// TIA Portal V17 export
// export: Created 2024-08-07T21:43:58.5559436Z, ExportSetting WithDefaults, DisplayName Totally Integrated Automation Portal, DisplayVersion V17 Update 7, DisplayName TIA Portal Openness, DisplayVersion V17 Update 7, DisplayName TIA Portal Version Control Interface, DisplayVersion V17, DisplayName SINAMICS Startdrive Advanced, DisplayVersion V17 SP2, DisplayName SINAMICS Startdrive G110M, G120, G120C, G120D, G120P, G115D, DisplayVersion V17 SP2, DisplayName SINAMICS Startdrive G130, G150, S120, S150, SINAMICS MV, S210, DisplayVersion V17 SP2, DisplayName STEP 7 Professional, DisplayVersion V17 Update 7, DisplayName STEP 7 Safety, DisplayVersion V17 Update 6, DisplayName WinCC Advanced / Unified PC, DisplayVersion V17 Update 7
FUNCTION "READERS" : Void   // FC19, LAD
{ S7_Optimized_Access := 'TRUE' }
VERSION : 0.1
// stored: AutoNumber true, IsIECCheckEnabled false, SetENOAutomatically false, UDAEnableTagReadback false
   VAR_TEMP
      done1 : Bool;
      done2 : Bool;
      done3 : Bool;
      done4 : Bool;
      ERROR_RECIBIDO_ESCANER_REAR_TUBE : Int;
      ERROR_RECIBIDO_ESCANER_FRONT_TUBE : Int;
      ERROR_RECIBIDO_ESCANER_LH_MEMBER : Int;
      ERROR_RECIBIDO_ESCANER_RH_MEMBER : Int;
   END_VAR
   VAR_TEMP   // added for the SCL form of the ladder/FBD networks
      _w1 : Bool;
   END_VAR
BEGIN

REGION Network 1: INIT
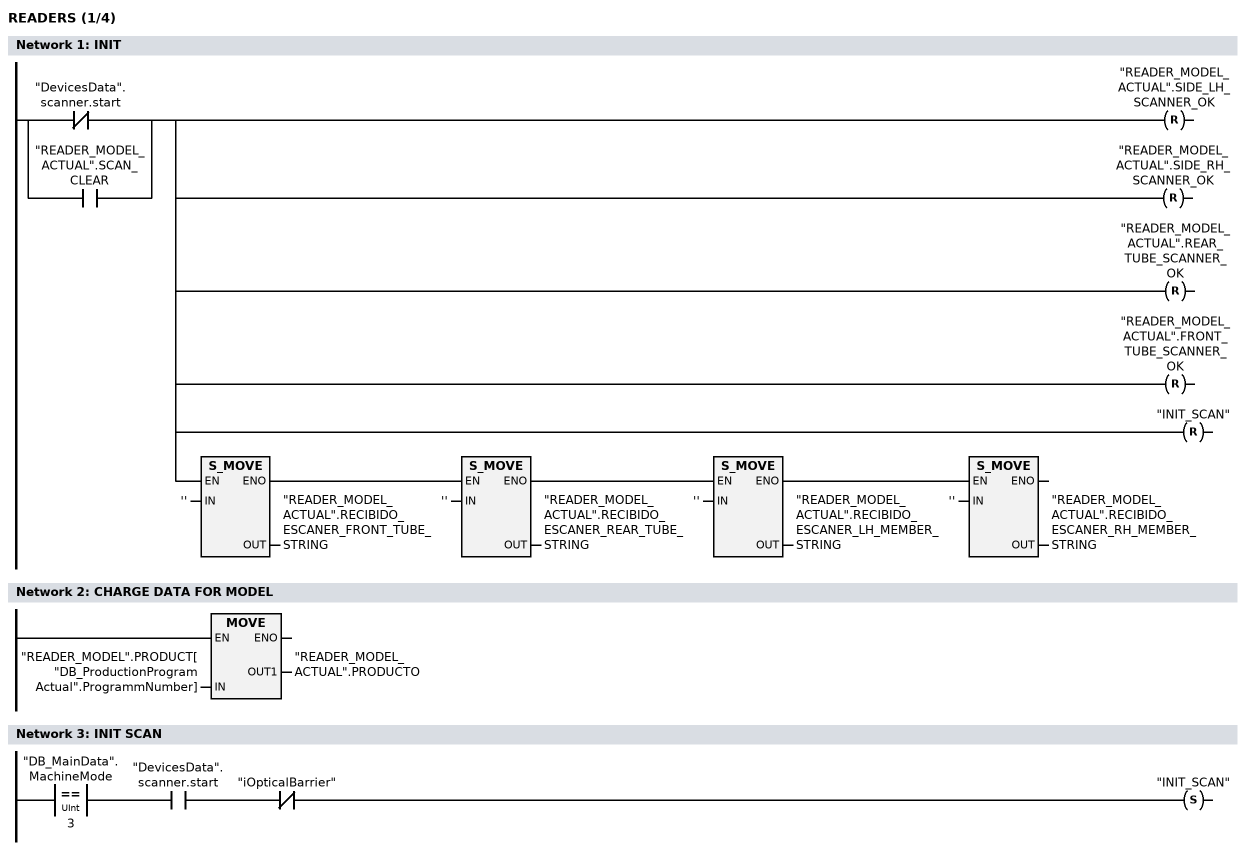
   RUNG wire#powerrail
      I_Contact( "DevicesData".scanner.start )
      wire#w1
      R_Coil( "READER_MODEL_ACTUAL".SIDE_LH_SCANNER_OK )
   END_RUNG
   RUNG wire#powerrail
      Contact( "READER_MODEL_ACTUAL".SCAN_CLEAR )
   END_RUNG wire#w1
   RUNG wire#w1
      R_Coil( "READER_MODEL_ACTUAL".SIDE_RH_SCANNER_OK )
   END_RUNG
   RUNG wire#w1
      R_Coil( "READER_MODEL_ACTUAL".REAR_TUBE_SCANNER_OK )
   END_RUNG
   RUNG wire#w1
      R_Coil( "READER_MODEL_ACTUAL".FRONT_TUBE_SCANNER_OK )
   END_RUNG
   RUNG wire#w1
      R_Coil( "INIT_SCAN" )
   END_RUNG
   RUNG wire#w1
      S_Move(in := '', out => "READER_MODEL_ACTUAL".RECIBIDO_ESCANER_FRONT_TUBE_STRING)
      S_Move(in := '', out => "READER_MODEL_ACTUAL".RECIBIDO_ESCANER_REAR_TUBE_STRING)
      S_Move(in := '', out => "READER_MODEL_ACTUAL".RECIBIDO_ESCANER_LH_MEMBER_STRING)
      S_Move(in := '', out => "READER_MODEL_ACTUAL".RECIBIDO_ESCANER_RH_MEMBER_STRING)
   END_RUNG
   // the same network as SCL:
   IF NOT "DevicesData".scanner.start OR "READER_MODEL_ACTUAL".SCAN_CLEAR THEN
       "READER_MODEL_ACTUAL".SIDE_LH_SCANNER_OK := FALSE;
       "READER_MODEL_ACTUAL".SIDE_RH_SCANNER_OK := FALSE;
       "READER_MODEL_ACTUAL".REAR_TUBE_SCANNER_OK := FALSE;
       "READER_MODEL_ACTUAL".FRONT_TUBE_SCANNER_OK := FALSE;
       "INIT_SCAN" := FALSE;
       "READER_MODEL_ACTUAL".RECIBIDO_ESCANER_FRONT_TUBE_STRING := '';
       "READER_MODEL_ACTUAL".RECIBIDO_ESCANER_REAR_TUBE_STRING := '';
       "READER_MODEL_ACTUAL".RECIBIDO_ESCANER_LH_MEMBER_STRING := '';
       "READER_MODEL_ACTUAL".RECIBIDO_ESCANER_RH_MEMBER_STRING := '';
   END_IF;
END_REGION

REGION Network 2: CHARGE DATA FOR MODEL
   RUNG wire#powerrail
      Move(in := "READER_MODEL".PRODUCT["DB_ProductionProgramActual".ProgrammNumber], out1 => "READER_MODEL_ACTUAL".PRODUCTO)
   END_RUNG
   // the same network as SCL:
   "READER_MODEL_ACTUAL".PRODUCTO := "READER_MODEL".PRODUCT["DB_ProductionProgramActual".ProgrammNumber];
END_REGION

REGION Network 3: INIT SCAN
   RUNG wire#powerrail
      { S7_Templates := "SrcType := UInt" } EQ_Contact(in1 := "DB_MainData".MachineMode, in2 := 3)
      Contact( "DevicesData".scanner.start )
      I_Contact( "iOpticalBarrier" )
      S_Coil( "INIT_SCAN" )
   END_RUNG
   // the same network as SCL:
   IF ("DB_MainData".MachineMode = 3) AND "DevicesData".scanner.start AND NOT "iOpticalBarrier" THEN
       "INIT_SCAN" := TRUE;
   END_IF;
END_REGION

REGION Network 4: LECTURA ESCANER REAR TUBE
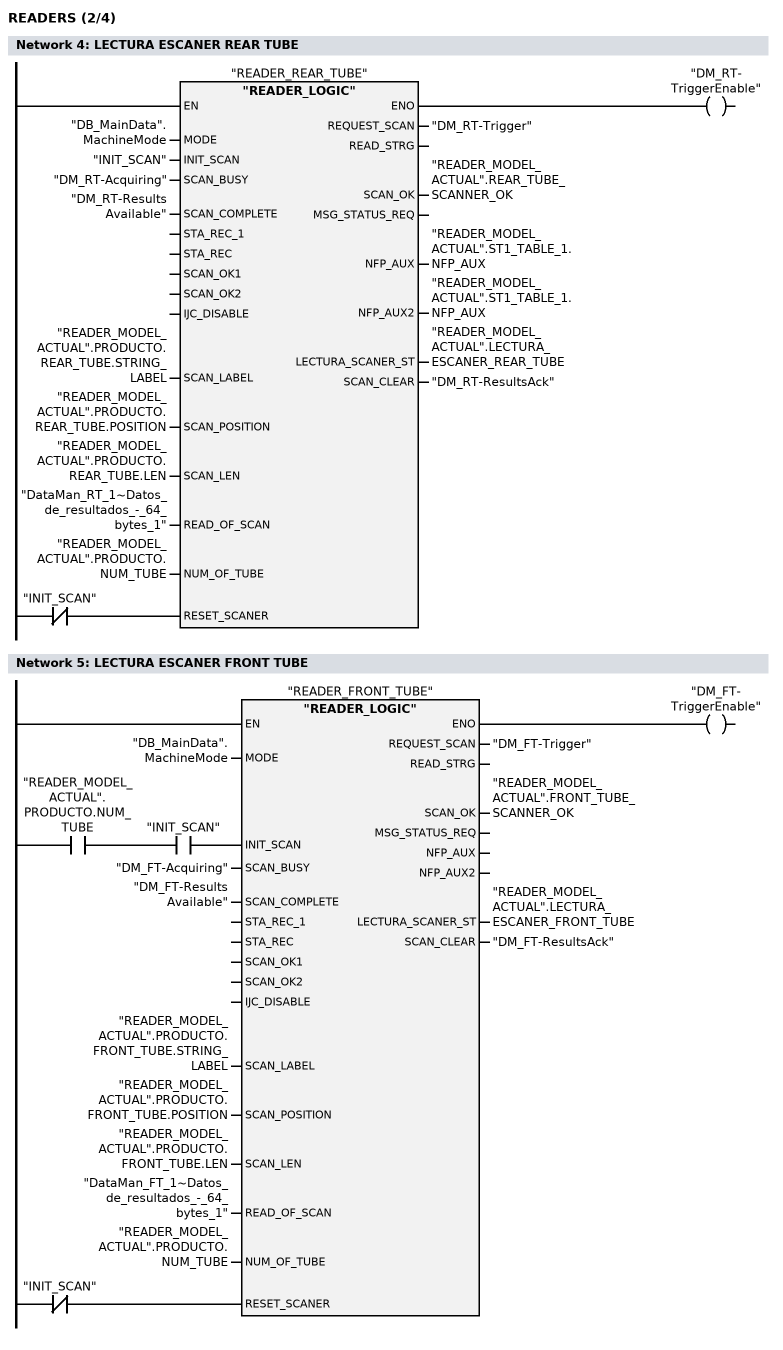
   RUNG wire#powerrail
      "READER_REAR_TUBE"(RESET_SCANER := wire#w1, MODE := "DB_MainData".MachineMode, INIT_SCAN := "INIT_SCAN", SCAN_BUSY := "DM_RT-Acquiring", SCAN_COMPLETE := "DM_RT-Results Available", STA_REC_1 :=, STA_REC :=, SCAN_OK1 :=, SCAN_OK2 :=, IJC_DISABLE :=, SCAN_LABEL := "READER_MODEL_ACTUAL".PRODUCTO.REAR_TUBE.STRING_LABEL, SCAN_POSITION := "READER_MODEL_ACTUAL".PRODUCTO.REAR_TUBE.POSITION, SCAN_LEN := "READER_MODEL_ACTUAL".PRODUCTO.REAR_TUBE.LEN, READ_OF_SCAN := "DataMan_RT_1~Datos_de_resultados_-_64_bytes_1", NUM_OF_TUBE := "READER_MODEL_ACTUAL".PRODUCTO.NUM_TUBE, REQUEST_SCAN => "DM_RT-Trigger", READ_STRG =>, SCAN_OK => "READER_MODEL_ACTUAL".REAR_TUBE_SCANNER_OK, MSG_STATUS_REQ =>, NFP_AUX => "READER_MODEL_ACTUAL".ST1_TABLE_1.NFP_AUX, NFP_AUX2 => "READER_MODEL_ACTUAL".ST1_TABLE_1.NFP_AUX, LECTURA_SCANER_ST => "READER_MODEL_ACTUAL".LECTURA_ESCANER_REAR_TUBE, SCAN_CLEAR => "DM_RT-ResultsAck")
      Coil( "DM_RT-TriggerEnable" )
   END_RUNG
   RUNG wire#powerrail
      I_Contact( "INIT_SCAN" )
   END_RUNG wire#w1
   // the same network as SCL:
   "READER_REAR_TUBE"(MODE := "DB_MainData".MachineMode,   // "READER_LOGIC"
                      INIT_SCAN := "INIT_SCAN",
                      SCAN_BUSY := "DM_RT-Acquiring",
                      SCAN_COMPLETE := "DM_RT-Results Available",
                      SCAN_LABEL := "READER_MODEL_ACTUAL".PRODUCTO.REAR_TUBE.STRING_LABEL,
                      SCAN_POSITION := "READER_MODEL_ACTUAL".PRODUCTO.REAR_TUBE.POSITION,
                      SCAN_LEN := "READER_MODEL_ACTUAL".PRODUCTO.REAR_TUBE.LEN,
                      READ_OF_SCAN := "DataMan_RT_1~Datos_de_resultados_-_64_bytes_1",
                      NUM_OF_TUBE := "READER_MODEL_ACTUAL".PRODUCTO.NUM_TUBE,
                      RESET_SCANER := NOT "INIT_SCAN",
                      REQUEST_SCAN => "DM_RT-Trigger",
                      SCAN_OK => "READER_MODEL_ACTUAL".REAR_TUBE_SCANNER_OK,
                      NFP_AUX => "READER_MODEL_ACTUAL".ST1_TABLE_1.NFP_AUX,
                      NFP_AUX2 => "READER_MODEL_ACTUAL".ST1_TABLE_1.NFP_AUX,
                      LECTURA_SCANER_ST => "READER_MODEL_ACTUAL".LECTURA_ESCANER_REAR_TUBE,
                      SCAN_CLEAR => "DM_RT-ResultsAck",
                      ENO => #_w1);
   "DM_RT-TriggerEnable" := #_w1;
END_REGION

REGION Network 5: LECTURA ESCANER FRONT TUBE
   RUNG wire#powerrail
      "READER_FRONT_TUBE"(INIT_SCAN := wire#w1, RESET_SCANER := wire#w2, MODE := "DB_MainData".MachineMode, SCAN_BUSY := "DM_FT-Acquiring", SCAN_COMPLETE := "DM_FT-Results Available", STA_REC_1 :=, STA_REC :=, SCAN_OK1 :=, SCAN_OK2 :=, IJC_DISABLE :=, SCAN_LABEL := "READER_MODEL_ACTUAL".PRODUCTO.FRONT_TUBE.STRING_LABEL, SCAN_POSITION := "READER_MODEL_ACTUAL".PRODUCTO.FRONT_TUBE.POSITION, SCAN_LEN := "READER_MODEL_ACTUAL".PRODUCTO.FRONT_TUBE.LEN, READ_OF_SCAN := "DataMan_FT_1~Datos_de_resultados_-_64_bytes_1", NUM_OF_TUBE := "READER_MODEL_ACTUAL".PRODUCTO.NUM_TUBE, REQUEST_SCAN => "DM_FT-Trigger", READ_STRG =>, SCAN_OK => "READER_MODEL_ACTUAL".FRONT_TUBE_SCANNER_OK, MSG_STATUS_REQ =>, NFP_AUX =>, NFP_AUX2 =>, LECTURA_SCANER_ST => "READER_MODEL_ACTUAL".LECTURA_ESCANER_FRONT_TUBE, SCAN_CLEAR => "DM_FT-ResultsAck")
      Coil( "DM_FT-TriggerEnable" )
   END_RUNG
   RUNG wire#powerrail
      Contact( "READER_MODEL_ACTUAL".PRODUCTO.NUM_TUBE )
      Contact( "INIT_SCAN" )
   END_RUNG wire#w1
   RUNG wire#powerrail
      I_Contact( "INIT_SCAN" )
   END_RUNG wire#w2
   // the same network as SCL:
   "READER_FRONT_TUBE"(MODE := "DB_MainData".MachineMode,   // "READER_LOGIC"
                       INIT_SCAN := "READER_MODEL_ACTUAL".PRODUCTO.NUM_TUBE AND "INIT_SCAN",
                       SCAN_BUSY := "DM_FT-Acquiring",
                       SCAN_COMPLETE := "DM_FT-Results Available",
                       SCAN_LABEL := "READER_MODEL_ACTUAL".PRODUCTO.FRONT_TUBE.STRING_LABEL,
                       SCAN_POSITION := "READER_MODEL_ACTUAL".PRODUCTO.FRONT_TUBE.POSITION,
                       SCAN_LEN := "READER_MODEL_ACTUAL".PRODUCTO.FRONT_TUBE.LEN,
                       READ_OF_SCAN := "DataMan_FT_1~Datos_de_resultados_-_64_bytes_1",
                       NUM_OF_TUBE := "READER_MODEL_ACTUAL".PRODUCTO.NUM_TUBE,
                       RESET_SCANER := NOT "INIT_SCAN",
                       REQUEST_SCAN => "DM_FT-Trigger",
                       SCAN_OK => "READER_MODEL_ACTUAL".FRONT_TUBE_SCANNER_OK,
                       LECTURA_SCANER_ST => "READER_MODEL_ACTUAL".LECTURA_ESCANER_FRONT_TUBE,
                       SCAN_CLEAR => "DM_FT-ResultsAck",
                       ENO => #_w1);
   "DM_FT-TriggerEnable" := #_w1;
END_REGION

REGION Network 6: LECTURA ESCANER SIDE LH
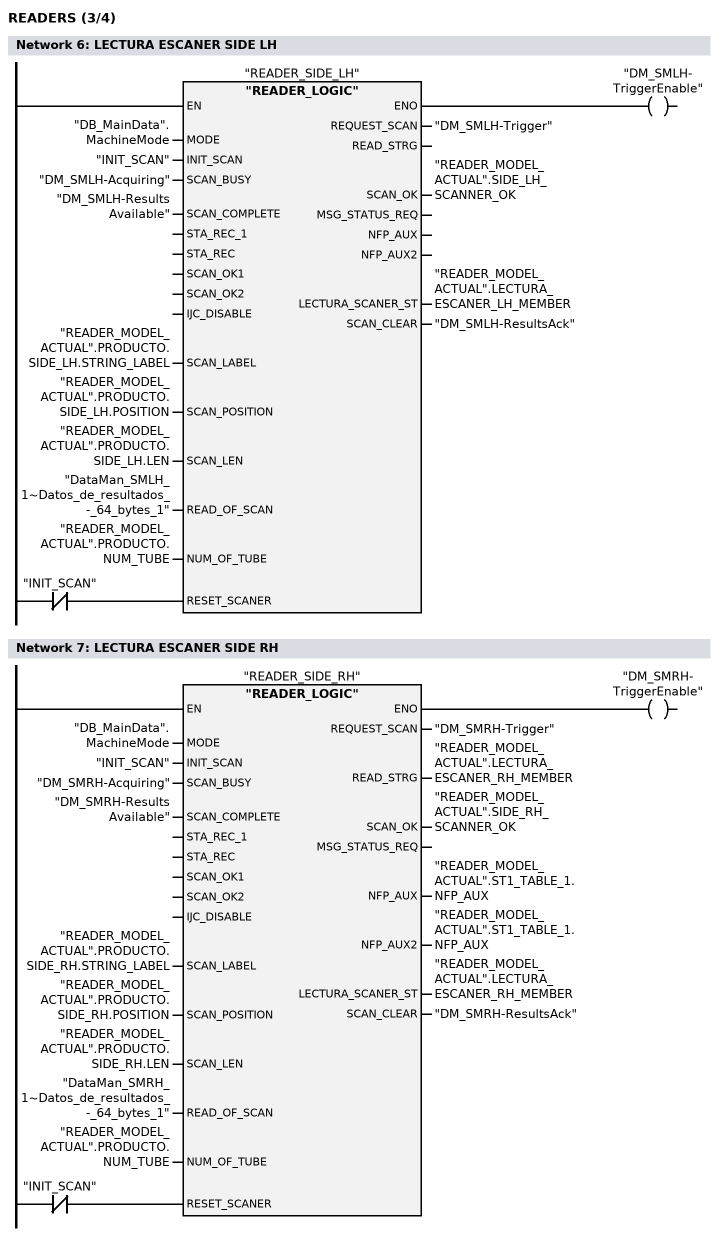
   RUNG wire#powerrail
      "READER_SIDE_LH"(RESET_SCANER := wire#w1, MODE := "DB_MainData".MachineMode, INIT_SCAN := "INIT_SCAN", SCAN_BUSY := "DM_SMLH-Acquiring", SCAN_COMPLETE := "DM_SMLH-Results Available", STA_REC_1 :=, STA_REC :=, SCAN_OK1 :=, SCAN_OK2 :=, IJC_DISABLE :=, SCAN_LABEL := "READER_MODEL_ACTUAL".PRODUCTO.SIDE_LH.STRING_LABEL, SCAN_POSITION := "READER_MODEL_ACTUAL".PRODUCTO.SIDE_LH.POSITION, SCAN_LEN := "READER_MODEL_ACTUAL".PRODUCTO.SIDE_LH.LEN, READ_OF_SCAN := "DataMan_SMLH_1~Datos_de_resultados_-_64_bytes_1", NUM_OF_TUBE := "READER_MODEL_ACTUAL".PRODUCTO.NUM_TUBE, REQUEST_SCAN => "DM_SMLH-Trigger", READ_STRG =>, SCAN_OK => "READER_MODEL_ACTUAL".SIDE_LH_SCANNER_OK, MSG_STATUS_REQ =>, NFP_AUX =>, NFP_AUX2 =>, LECTURA_SCANER_ST => "READER_MODEL_ACTUAL".LECTURA_ESCANER_LH_MEMBER, SCAN_CLEAR => "DM_SMLH-ResultsAck")
      Coil( "DM_SMLH-TriggerEnable" )
   END_RUNG
   RUNG wire#powerrail
      I_Contact( "INIT_SCAN" )
   END_RUNG wire#w1
   // the same network as SCL:
   "READER_SIDE_LH"(MODE := "DB_MainData".MachineMode,   // "READER_LOGIC"
                    INIT_SCAN := "INIT_SCAN",
                    SCAN_BUSY := "DM_SMLH-Acquiring",
                    SCAN_COMPLETE := "DM_SMLH-Results Available",
                    SCAN_LABEL := "READER_MODEL_ACTUAL".PRODUCTO.SIDE_LH.STRING_LABEL,
                    SCAN_POSITION := "READER_MODEL_ACTUAL".PRODUCTO.SIDE_LH.POSITION,
                    SCAN_LEN := "READER_MODEL_ACTUAL".PRODUCTO.SIDE_LH.LEN,
                    READ_OF_SCAN := "DataMan_SMLH_1~Datos_de_resultados_-_64_bytes_1",
                    NUM_OF_TUBE := "READER_MODEL_ACTUAL".PRODUCTO.NUM_TUBE,
                    RESET_SCANER := NOT "INIT_SCAN",
                    REQUEST_SCAN => "DM_SMLH-Trigger",
                    SCAN_OK => "READER_MODEL_ACTUAL".SIDE_LH_SCANNER_OK,
                    LECTURA_SCANER_ST => "READER_MODEL_ACTUAL".LECTURA_ESCANER_LH_MEMBER,
                    SCAN_CLEAR => "DM_SMLH-ResultsAck",
                    ENO => #_w1);
   "DM_SMLH-TriggerEnable" := #_w1;
END_REGION

REGION Network 7: LECTURA ESCANER SIDE RH
   RUNG wire#powerrail
      "READER_SIDE_RH"(RESET_SCANER := wire#w1, MODE := "DB_MainData".MachineMode, INIT_SCAN := "INIT_SCAN", SCAN_BUSY := "DM_SMRH-Acquiring", SCAN_COMPLETE := "DM_SMRH-Results Available", STA_REC_1 :=, STA_REC :=, SCAN_OK1 :=, SCAN_OK2 :=, IJC_DISABLE :=, SCAN_LABEL := "READER_MODEL_ACTUAL".PRODUCTO.SIDE_RH.STRING_LABEL, SCAN_POSITION := "READER_MODEL_ACTUAL".PRODUCTO.SIDE_RH.POSITION, SCAN_LEN := "READER_MODEL_ACTUAL".PRODUCTO.SIDE_RH.LEN, READ_OF_SCAN := "DataMan_SMRH_1~Datos_de_resultados_-_64_bytes_1", NUM_OF_TUBE := "READER_MODEL_ACTUAL".PRODUCTO.NUM_TUBE, REQUEST_SCAN => "DM_SMRH-Trigger", READ_STRG => "READER_MODEL_ACTUAL".LECTURA_ESCANER_RH_MEMBER, SCAN_OK => "READER_MODEL_ACTUAL".SIDE_RH_SCANNER_OK, MSG_STATUS_REQ =>, NFP_AUX => "READER_MODEL_ACTUAL".ST1_TABLE_1.NFP_AUX, NFP_AUX2 => "READER_MODEL_ACTUAL".ST1_TABLE_1.NFP_AUX, LECTURA_SCANER_ST => "READER_MODEL_ACTUAL".LECTURA_ESCANER_RH_MEMBER, SCAN_CLEAR => "DM_SMRH-ResultsAck")
      Coil( "DM_SMRH-TriggerEnable" )
   END_RUNG
   RUNG wire#powerrail
      I_Contact( "INIT_SCAN" )
   END_RUNG wire#w1
   // the same network as SCL:
   "READER_SIDE_RH"(MODE := "DB_MainData".MachineMode,   // "READER_LOGIC"
                    INIT_SCAN := "INIT_SCAN",
                    SCAN_BUSY := "DM_SMRH-Acquiring",
                    SCAN_COMPLETE := "DM_SMRH-Results Available",
                    SCAN_LABEL := "READER_MODEL_ACTUAL".PRODUCTO.SIDE_RH.STRING_LABEL,
                    SCAN_POSITION := "READER_MODEL_ACTUAL".PRODUCTO.SIDE_RH.POSITION,
                    SCAN_LEN := "READER_MODEL_ACTUAL".PRODUCTO.SIDE_RH.LEN,
                    READ_OF_SCAN := "DataMan_SMRH_1~Datos_de_resultados_-_64_bytes_1",
                    NUM_OF_TUBE := "READER_MODEL_ACTUAL".PRODUCTO.NUM_TUBE,
                    RESET_SCANER := NOT "INIT_SCAN",
                    REQUEST_SCAN => "DM_SMRH-Trigger",
                    READ_STRG => "READER_MODEL_ACTUAL".LECTURA_ESCANER_RH_MEMBER,
                    SCAN_OK => "READER_MODEL_ACTUAL".SIDE_RH_SCANNER_OK,
                    NFP_AUX => "READER_MODEL_ACTUAL".ST1_TABLE_1.NFP_AUX,
                    NFP_AUX2 => "READER_MODEL_ACTUAL".ST1_TABLE_1.NFP_AUX,
                    LECTURA_SCANER_ST => "READER_MODEL_ACTUAL".LECTURA_ESCANER_RH_MEMBER,
                    SCAN_CLEAR => "DM_SMRH-ResultsAck",
                    ENO => #_w1);
   "DM_SMRH-TriggerEnable" := #_w1;
END_REGION

REGION Network 8: ALL SCANER OK
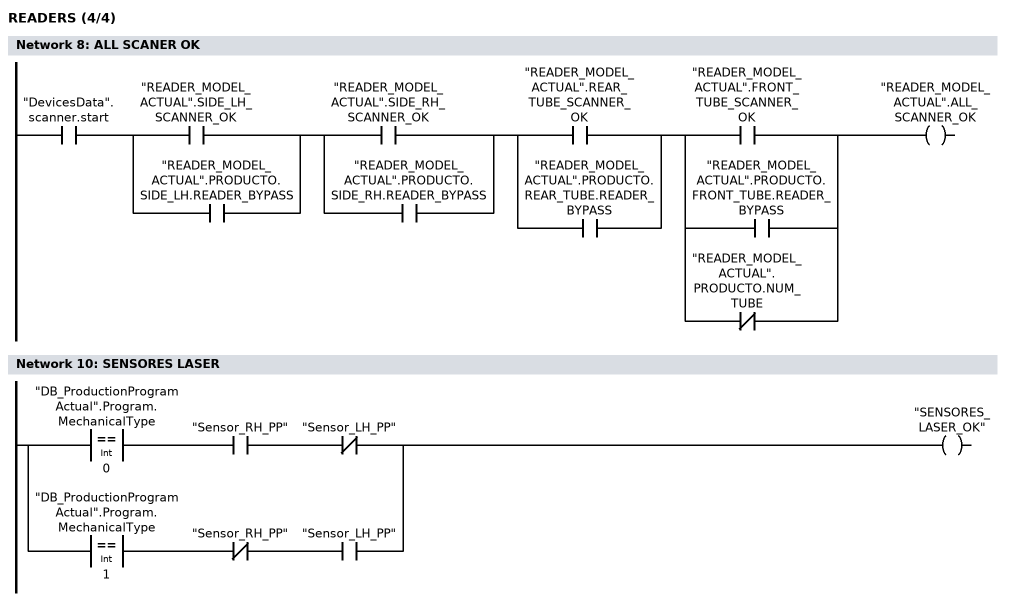
   RUNG wire#powerrail
      Contact( "DevicesData".scanner.start )
      wire#w1
      Contact( "READER_MODEL_ACTUAL".SIDE_LH_SCANNER_OK )
      wire#w2
      Contact( "READER_MODEL_ACTUAL".SIDE_RH_SCANNER_OK )
      wire#w3
      Contact( "READER_MODEL_ACTUAL".REAR_TUBE_SCANNER_OK )
      wire#w4
      Contact( "READER_MODEL_ACTUAL".FRONT_TUBE_SCANNER_OK )
      wire#w5
      Coil( "READER_MODEL_ACTUAL".ALL_SCANNER_OK )
   END_RUNG
   RUNG wire#w1
      Contact( "READER_MODEL_ACTUAL".PRODUCTO.SIDE_LH.READER_BYPASS )
   END_RUNG wire#w2
   RUNG wire#w2
      Contact( "READER_MODEL_ACTUAL".PRODUCTO.SIDE_RH.READER_BYPASS )
   END_RUNG wire#w3
   RUNG wire#w3
      Contact( "READER_MODEL_ACTUAL".PRODUCTO.REAR_TUBE.READER_BYPASS )
   END_RUNG wire#w4
   RUNG wire#w4
      Contact( "READER_MODEL_ACTUAL".PRODUCTO.FRONT_TUBE.READER_BYPASS )
   END_RUNG wire#w5
   RUNG wire#w4
      I_Contact( "READER_MODEL_ACTUAL".PRODUCTO.NUM_TUBE )
   END_RUNG wire#w5
   // the same network as SCL:
   "READER_MODEL_ACTUAL".ALL_SCANNER_OK := "DevicesData".scanner.start AND ("READER_MODEL_ACTUAL".SIDE_LH_SCANNER_OK OR "READER_MODEL_ACTUAL".PRODUCTO.SIDE_LH.READER_BYPASS) AND ("READER_MODEL_ACTUAL".SIDE_RH_SCANNER_OK OR "READER_MODEL_ACTUAL".PRODUCTO.SIDE_RH.READER_BYPASS) AND ("READER_MODEL_ACTUAL".REAR_TUBE_SCANNER_OK OR "READER_MODEL_ACTUAL".PRODUCTO.REAR_TUBE.READER_BYPASS) AND ("READER_MODEL_ACTUAL".FRONT_TUBE_SCANNER_OK OR "READER_MODEL_ACTUAL".PRODUCTO.FRONT_TUBE.READER_BYPASS OR NOT "READER_MODEL_ACTUAL".PRODUCTO.NUM_TUBE);
END_REGION

REGION Network 9: SEND TRC 1 MSG5
END_REGION

REGION Network 10: SENSORES LASER
   RUNG wire#powerrail
      { S7_Templates := "SrcType := Int" } EQ_Contact(in1 := "DB_ProductionProgramActual".Program.MechanicalType, in2 := 0)
      Contact( "Sensor_RH_PP" )
      I_Contact( "Sensor_LH_PP" )
      wire#w1
      Coil( "SENSORES_LASER_OK" )
   END_RUNG
   RUNG wire#powerrail
      { S7_Templates := "SrcType := Int" } EQ_Contact(in1 := "DB_ProductionProgramActual".Program.MechanicalType, in2 := 1)
      I_Contact( "Sensor_RH_PP" )
      Contact( "Sensor_LH_PP" )
   END_RUNG wire#w1
   // the same network as SCL:
   "SENSORES_LASER_OK" := (("DB_ProductionProgramActual".Program.MechanicalType = 0) AND "Sensor_RH_PP" AND NOT "Sensor_LH_PP") OR (("DB_ProductionProgramActual".Program.MechanicalType = 1) AND NOT "Sensor_RH_PP" AND "Sensor_LH_PP");
END_REGION
END_FUNCTION
